// Mitsubishi GX Works2 project: סופי   PLC: FX3G

// global labels: Global1
VAR_GLOBAL
  input_sw AT M0 : BOOL;
  active_day AT M7 : BOOL;
  work_day AT X010 : BOOL;
  flour_stock AT D1100 : REAL;
  flour_input AT D1110 : REAL;
  yeast_stock AT D1120 : REAL;
  oil_stock AT D1160 : REAL;
  spices_stock AT D1180 : REAL;
  yeast_input AT D1130 : REAL;
  water_input AT D1150 : REAL;
  water_stock AT D1140 : REAL;
  oil_input AT D1170 : REAL;
  spices_input AT D1190 : REAL;
  check_flour AT M1 : BOOL;
END_VAR
VAR_GLOBAL CONSTANT
  min_flour_stock : REAL := 100.0;
  yeast_con : REAL := 0.2;
END_VAR
VAR_GLOBAL
  save_mul AT D1200 : REAL;
  check_yeast AT M2 : BOOL;
END_VAR
VAR_GLOBAL CONSTANT
  water_con : REAL := 0.5;
END_VAR
VAR_GLOBAL
  check_water AT M3 : BOOL;
END_VAR
VAR_GLOBAL CONSTANT
  oil_con : REAL := 0.3;
END_VAR
VAR_GLOBAL
  stock_stock AT D1160 : REAL;
  check_oil AT M4 : BOOL;
END_VAR
VAR_GLOBAL CONSTANT
  spices_con : REAL := 0.1;
END_VAR
VAR_GLOBAL
  check_spices AT M5 : BOOL;
  check_stock AT M6 : BOOL;
  emergency_sw AT X007 : BOOL;
END_VAR
VAR_GLOBAL CONSTANT
  flicker_time : INT := 5;
  flicker_con : INT := 6;
  flicker_timer : INT := 30;
  flick_time : INT := 5;
END_VAR
VAR_GLOBAL
  start_dough AT X001 : BOOL;
END_VAR
VAR_GLOBAL CONSTANT
  sec : INT := 30;
END_VAR
VAR_GLOBAL
  end_dough AT TS194 : BOOL;
  dough_light AT Y001 : BOOL;
END_VAR
VAR_GLOBAL CONSTANT
  flour_q : REAL := 100.0;
  yeast_q : REAL := 20.0;
  water_q : REAL := 50.0;
  oil_q : REAL := 30.0;
  spices_q : REAL := 10.0;
END_VAR
VAR_GLOBAL
  active_day_bulb AT Y010 : BOOL;
  start_ingridients_prep AT X002 : BOOL;
  ingridients_light AT Y005 : BOOL;
  start_swell AT X011 : BOOL;
  X11_COUNTER AT CC1 : BOOL;
END_VAR
VAR_GLOBAL CONSTANT
  X11_VAL : INT := 2;
END_VAR
VAR_GLOBAL
  swelling_time AT M8 : BOOL;
  swelling_light_timer AT TC195 : BOOL;
END_VAR
VAR_GLOBAL CONSTANT
  swelling_timer : INT := 30;
END_VAR
VAR_GLOBAL
  blink_light AT M9 : BOOL;
  blink3 AT TC3 : BOOL;
END_VAR
VAR_GLOBAL CONSTANT
  blink_time : INT := 5;
END_VAR
VAR_GLOBAL
  blink_timer3 AT TS3 : BOOL;
  blink_light3 AT Y002 : BOOL;
  blink4 AT TC4 : BOOL;
  blink_timer4 AT TS4 : BOOL;
  blink_light4 AT Y003 : BOOL;
  baking_timer AT TS5 : BOOL;
END_VAR
VAR_GLOBAL CONSTANT
  baking_time : INT := 40;
END_VAR
VAR_GLOBAL
  baking AT TC5 : BOOL;
  baking_light AT Y004 : BOOL;
  sample_quality AT X003 : BOOL;
  analog_input_2 AT D8281 : INT;
  save_analog_input_2 AT D1300 : INT;
END_VAR
VAR_GLOBAL CONSTANT
  lower_analog_bound : INT := K400;
  upper_analog_bound : INT := K2000;
END_VAR
VAR_GLOBAL
  good_quality AT M10 : BOOL;
  move_to_shelves_light AT Y006 : BOOL;
  move_to_shelves AT TC6 : BOOL;
END_VAR
VAR_GLOBAL CONSTANT
  move_to_shelves_time : INT := 50;
END_VAR
VAR_GLOBAL
  move_to_shelves_timer AT TS6 : BOOL;
  failure_counter AT CC2 : BOOL;
END_VAR
VAR_GLOBAL CONSTANT
  failure : INT := 2;
END_VAR
VAR_GLOBAL
  failure_count AT CS2 : BOOL;
  timer_flicker_light AT TC7 : BOOL;
END_VAR
VAR_GLOBAL CONSTANT
  flicker_duration : INT := 30;
END_VAR
VAR_GLOBAL
  timer_flicker1 AT TC8 : BOOL;
END_VAR
VAR_GLOBAL CONSTANT
  flicker_con1 : INT := 5;
END_VAR
VAR_GLOBAL
  timer_flicker2 AT TC9 : BOOL;
  timer_flicker_light_con AT TS7 : BOOL;
  timer_flicker2_con AT TS9 : BOOL;
  timer_flicker1_con AT TS8 : BOOL;
  M_11 AT M11 : BOOL;
  M_12 AT M12 : BOOL;
  flour_container AT D1210 : REAL;
  yeast_container AT D1220 : REAL;
  water_container AT D1230 : REAL;
  oil_container AT D1240 : REAL;
  spices_container AT D1250 : REAL;
  mixer AT D1260 : REAL;
END_VAR
VAR_GLOBAL CONSTANT
  on_sign : REAL := 1.0;
END_VAR
VAR_GLOBAL
  swelling_container AT D1270 : REAL;
  swelling_timer_s AT TS195 : BOOL;
  baking_pan AT D1280 : REAL;
  shelves AT D1290 : REAL;
  is_greater AT M26 : BOOL;
  finish_day AT M30 : BOOL;
  M_31 AT M31 : BOOL;
  M_32 AT M32 : BOOL;
  valid_x11 AT CS1 : BOOL;
  is_lower AT M27 : BOOL;
  finish_iteration AT M40 : BOOL;
  flicker_c AT CC0 : BOOL;
  timer3 AT TC194 : BOOL;
END_VAR

// task Task_01 (event TRUE, interval 0, priority 31): POU_01

PROGRAM POU_01
(* structured ladder/FBD written out as ST: instructions are called as NAME(EN, inputs, outputs); _pN, _eN, _tN stand for wires *)
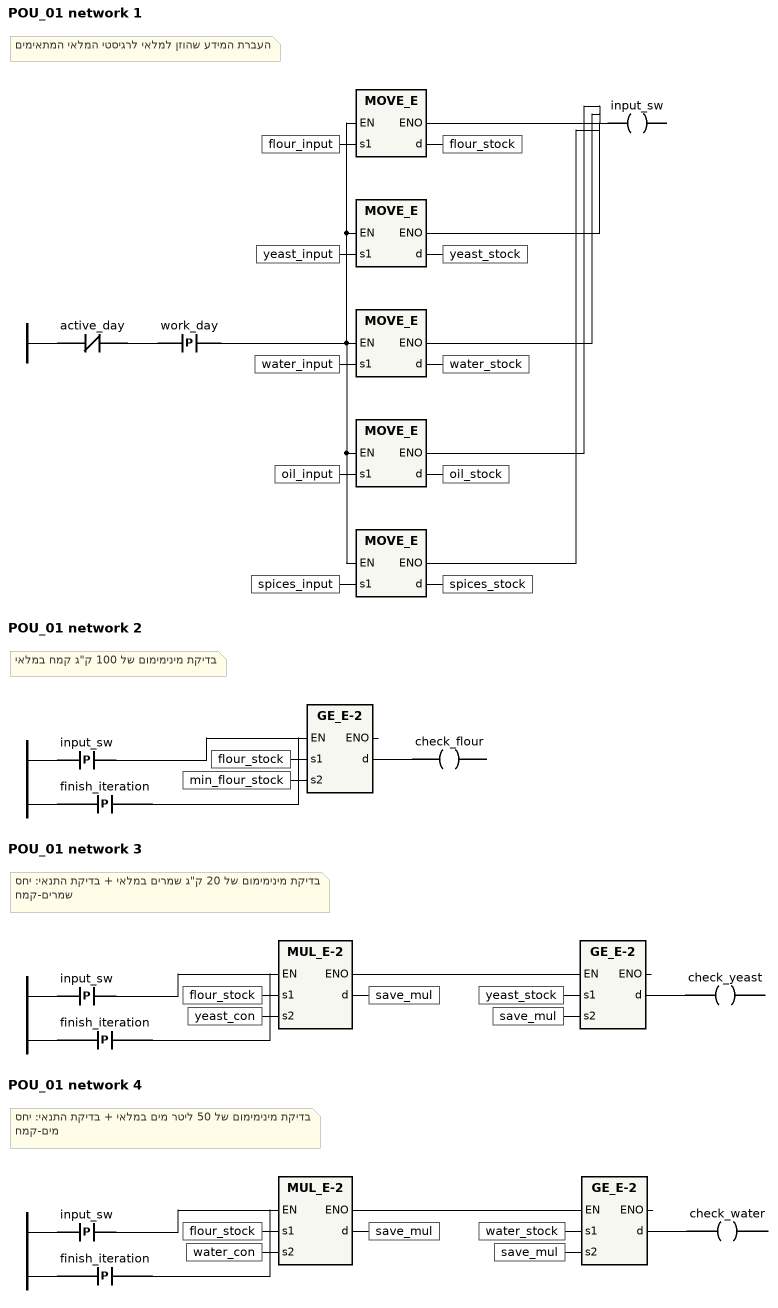
(* network 1 *)
(* העברת המידע שהוזן למלאי לרגיסטי המלאי המתאימים *)
_p1 := NOT active_day AND LDP(TRUE, work_day);
_e2 := MOVE_E(_p1, flour_input, flour_stock);
_e3 := MOVE_E(_p1, yeast_input, yeast_stock);
_e4 := MOVE_E(_p1, water_input, water_stock);
_e5 := MOVE_E(_p1, oil_input, oil_stock);
_e6 := MOVE_E(_p1, spices_input, spices_stock);
input_sw := _e2 OR _e3 OR _e4 OR _e5 OR _e6;
(* network 2 *)
(* בדיקת מינימימום של 100 ק"ג קמח במלאי *)
GE_E(LDP(TRUE, input_sw) OR LDP(TRUE, finish_iteration), flour_stock, min_flour_stock, _t1);
check_flour := _t1;
(* network 3 *)
(* בדיקת מינימימום של 20 ק"ג שמרים במלאי + בדיקת התנאי: יחס שמרים-קמח *)
_e1 := MUL_E(LDP(TRUE, input_sw) OR LDP(TRUE, finish_iteration), flour_stock, yeast_con, save_mul);
GE_E(_e1, yeast_stock, save_mul, _t2);
check_yeast := _t2;
(* network 4 *)
(* בדיקת מינימימום של 50 ליטר מים במלאי + בדיקת התנאי: יחס מים-קמח *)
_e1 := MUL_E(LDP(TRUE, input_sw) OR LDP(TRUE, finish_iteration), flour_stock, water_con, save_mul);
GE_E(_e1, water_stock, save_mul, _t2);
check_water := _t2;
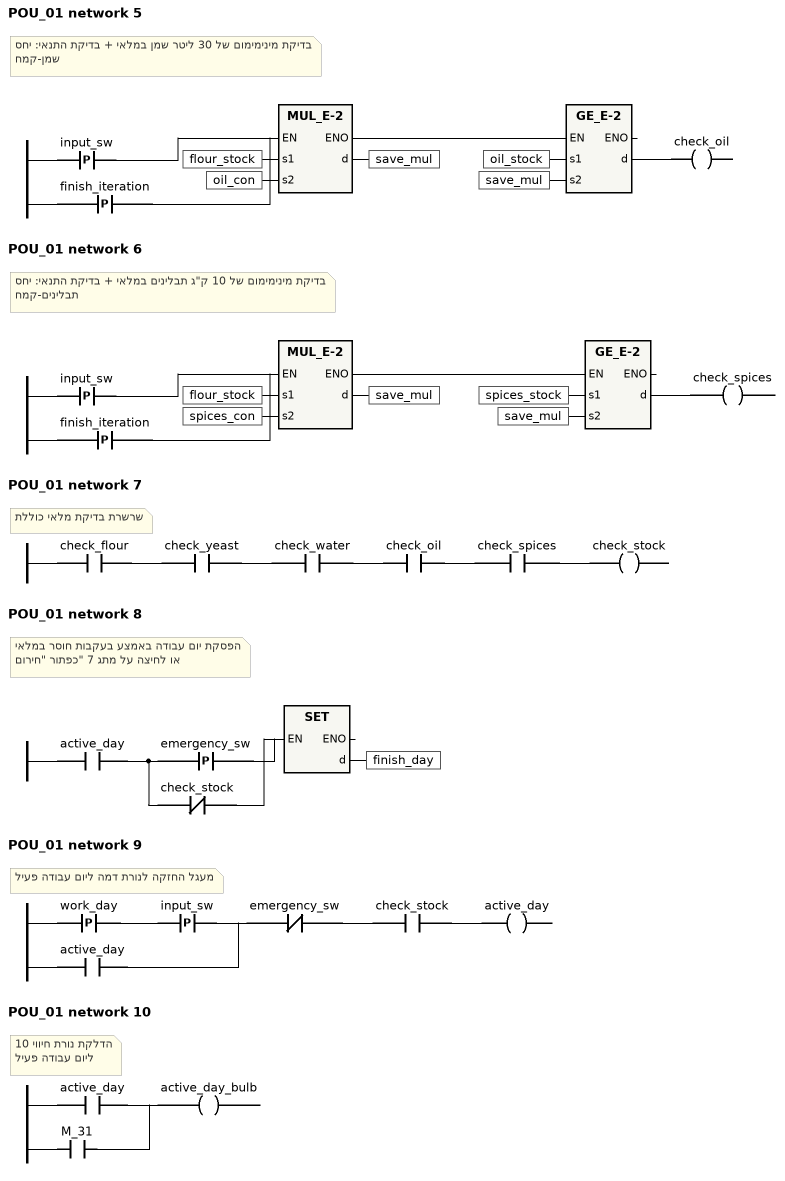
(* network 5 *)
(* בדיקת מינימימום של 30 ליטר שמן במלאי + בדיקת התנאי: יחס שמן-קמח *)
_e1 := MUL_E(LDP(TRUE, input_sw) OR LDP(TRUE, finish_iteration), flour_stock, oil_con, save_mul);
GE_E(_e1, oil_stock, save_mul, _t2);
check_oil := _t2;
(* network 6 *)
(* בדיקת מינימימום של 10 ק"ג תבלינים במלאי + בדיקת התנאי: יחס תבלינים-קמח *)
_e1 := MUL_E(LDP(TRUE, input_sw) OR LDP(TRUE, finish_iteration), flour_stock, spices_con, save_mul);
GE_E(_e1, spices_stock, save_mul, _t2);
check_spices := _t2;
(* network 7 *)
(* שרשרת בדיקת מלאי כוללת *)
check_stock := check_flour AND check_yeast AND check_water AND check_oil AND check_spices;
(* network 8 *)
(* הפסקת יום עבודה באמצע בעקבות חוסר במלאי / או לחיצה על מתג 7 "כפתור "חירום *)
SET((active_day AND LDP(TRUE, emergency_sw)) OR (active_day AND NOT check_stock), finish_day);
(* network 9 *)
(* מעגל החזקה לנורת דמה ליום עבודה פעיל *)
active_day := (((LDP(TRUE, work_day) AND LDP(TRUE, input_sw)) OR active_day) AND NOT emergency_sw) AND check_stock;
(* network 10 *)
(* הדלקת נורת חיווי 10 /  ליום עבודה פעיל *)
active_day_bulb := active_day OR M_31;
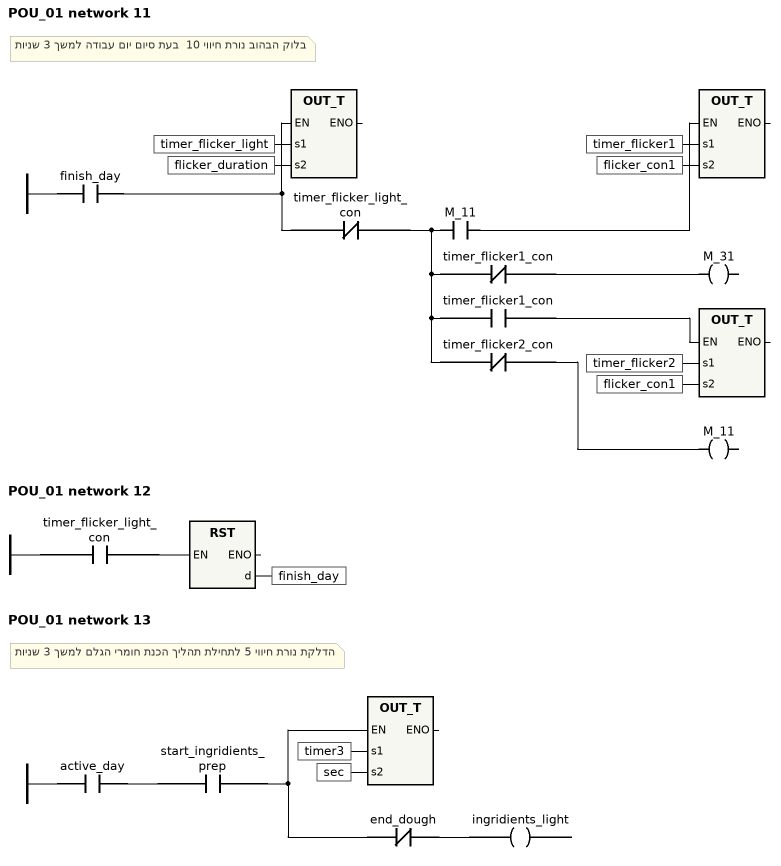
(* network 11 *)
(* בלוק הבהוב נורת חיווי 10  בעת סיום יום עבודה למשך 3 שניות *)
OUT_T(finish_day, timer_flicker_light, flicker_duration);
_p1 := finish_day AND NOT timer_flicker_light_con;
OUT_T(_p1 AND M_11, timer_flicker1, flicker_con1);
M_31 := _p1 AND NOT timer_flicker1_con;
OUT_T(_p1 AND timer_flicker1_con, timer_flicker2, flicker_con1);
M_11 := _p1 AND NOT timer_flicker2_con;
(* network 12 *)
RST(timer_flicker_light_con, finish_day);
(* network 13 *)
(* הדלקת נורת חיווי 5 לתחילת תהליך הכנת חומרי הגלם למשך 3 שניות *)
_p1 := active_day AND start_ingridients_prep;
OUT_T(_p1, timer3, sec);
ingridients_light := _p1 AND NOT end_dough;
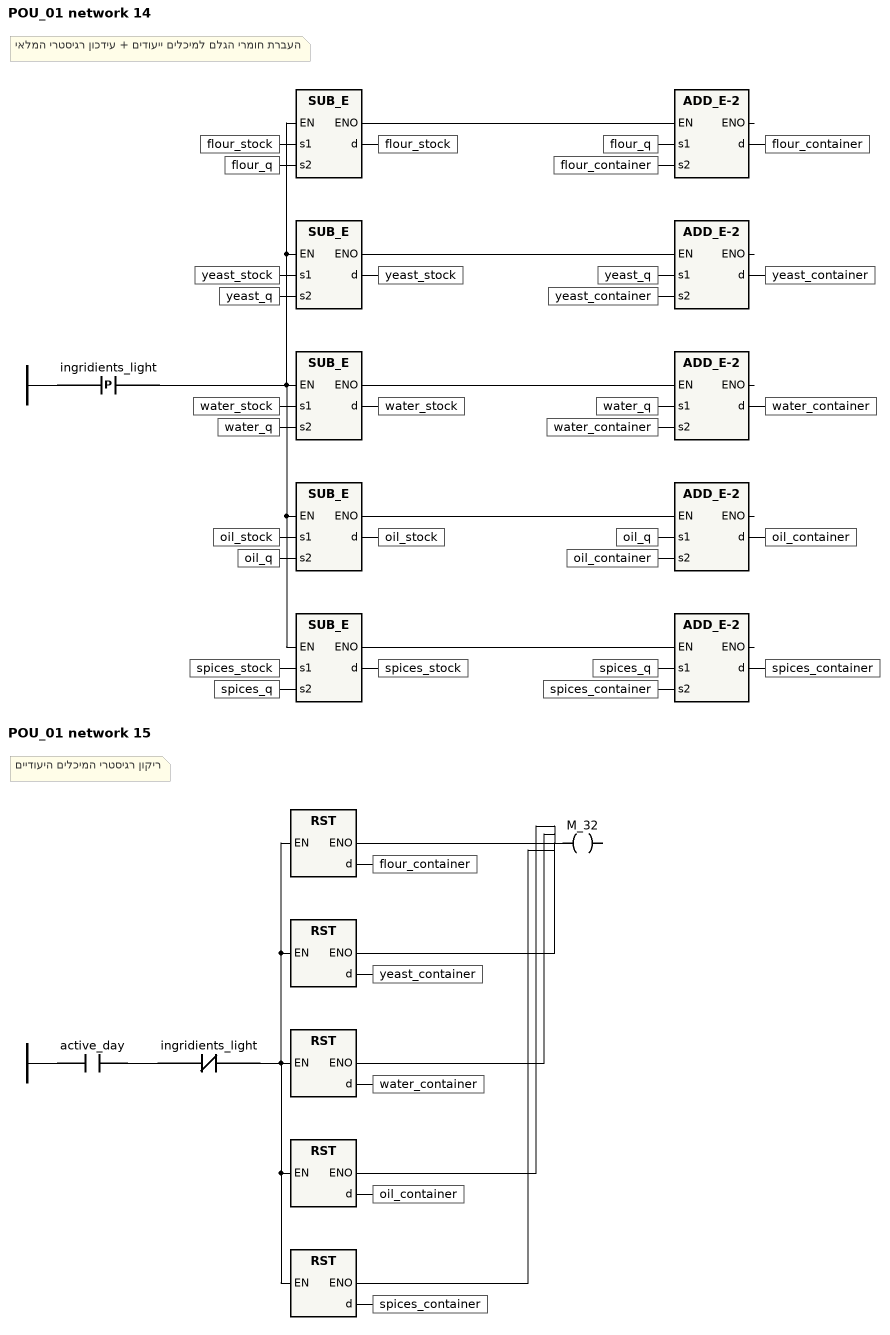
(* network 14 *)
(* העברת חומרי הגלם למיכלים ייעודים + עידכון רגיסטרי המלאי *)
_p1 := LDP(TRUE, ingridients_light);
_e2 := SUB_E(_p1, flour_stock, flour_q, flour_stock);
ADD_E(_e2, flour_q, flour_container, flour_container);
_e3 := SUB_E(_p1, yeast_stock, yeast_q, yeast_stock);
ADD_E(_e3, yeast_q, yeast_container, yeast_container);
_e4 := SUB_E(_p1, water_stock, water_q, water_stock);
ADD_E(_e4, water_q, water_container, water_container);
_e5 := SUB_E(_p1, oil_stock, oil_q, oil_stock);
ADD_E(_e5, oil_q, oil_container, oil_container);
_e6 := SUB_E(_p1, spices_stock, spices_q, spices_stock);
ADD_E(_e6, spices_q, spices_container, spices_container);
(* network 15 *)
(* ריקון רגיסטרי המיכלים היעודיים *)
_p1 := active_day AND NOT ingridients_light;
_e2 := RST(_p1, flour_container);
_e3 := RST(_p1, yeast_container);
_e4 := RST(_p1, water_container);
_e5 := RST(_p1, oil_container);
_e6 := RST(_p1, spices_container);
M_32 := _e2 OR _e3 OR _e4 OR _e5 OR _e6;
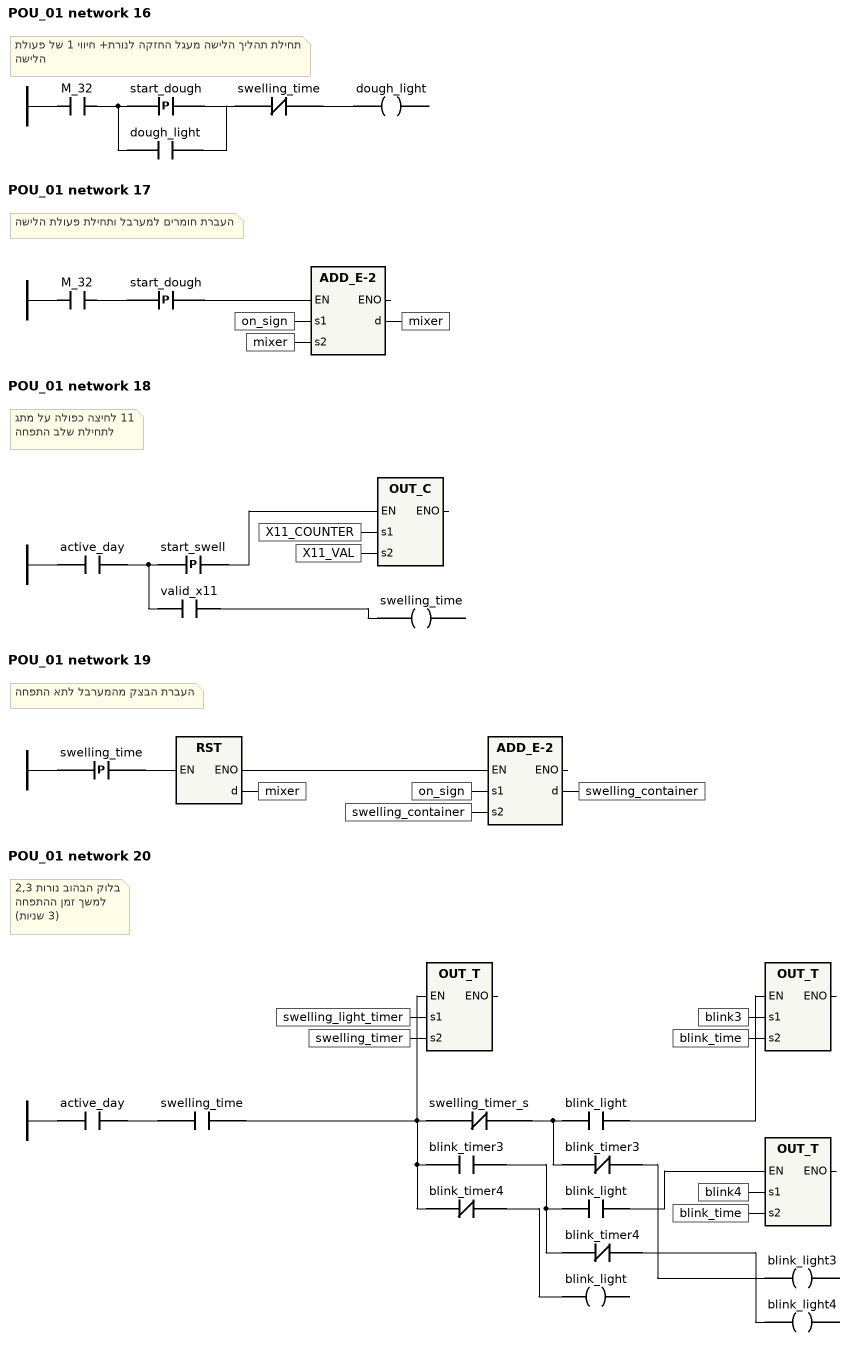
(* network 16 *)
(* תחילת תהליך הלישה מעגל החזקה לנורת+ חיווי 1 של פעולת הלישה *)
dough_light := ((M_32 AND LDP(TRUE, start_dough)) OR (M_32 AND dough_light)) AND NOT swelling_time;
(* network 17 *)
(* העברת חומרים למערבל ותחילת פעולת הלישה *)
ADD_E(M_32 AND LDP(TRUE, start_dough), on_sign, mixer, mixer);
(* network 18 *)
(* 11 לחיצה כפולה על מתג  / לתחילת שלב התפחה *)
OUT_C(active_day AND LDP(TRUE, start_swell), X11_COUNTER, X11_VAL);
swelling_time := active_day AND valid_x11;
(* network 19 *)
(* העברת הבצק מהמערבל לתא התפחה *)
_e1 := RST(LDP(TRUE, swelling_time), mixer);
ADD_E(_e1, on_sign, swelling_container, swelling_container);
(* network 20 *)
(* בלוק הבהוב נורות 2,3 /  למשך זמן ההתפחה /  (3 שניות) *)
_p1 := active_day AND swelling_time;
OUT_T(_p1, swelling_light_timer, swelling_timer);
_p2 := _p1 AND NOT swelling_timer_s;
OUT_T(_p2 AND blink_light, blink3, blink_time);
blink_light3 := _p2 AND NOT blink_timer3;
_p3 := _p1 AND blink_timer3;
OUT_T(_p3 AND blink_light, blink4, blink_time);
blink_light4 := _p3 AND NOT blink_timer4;
blink_light := _p1 AND NOT blink_timer4;
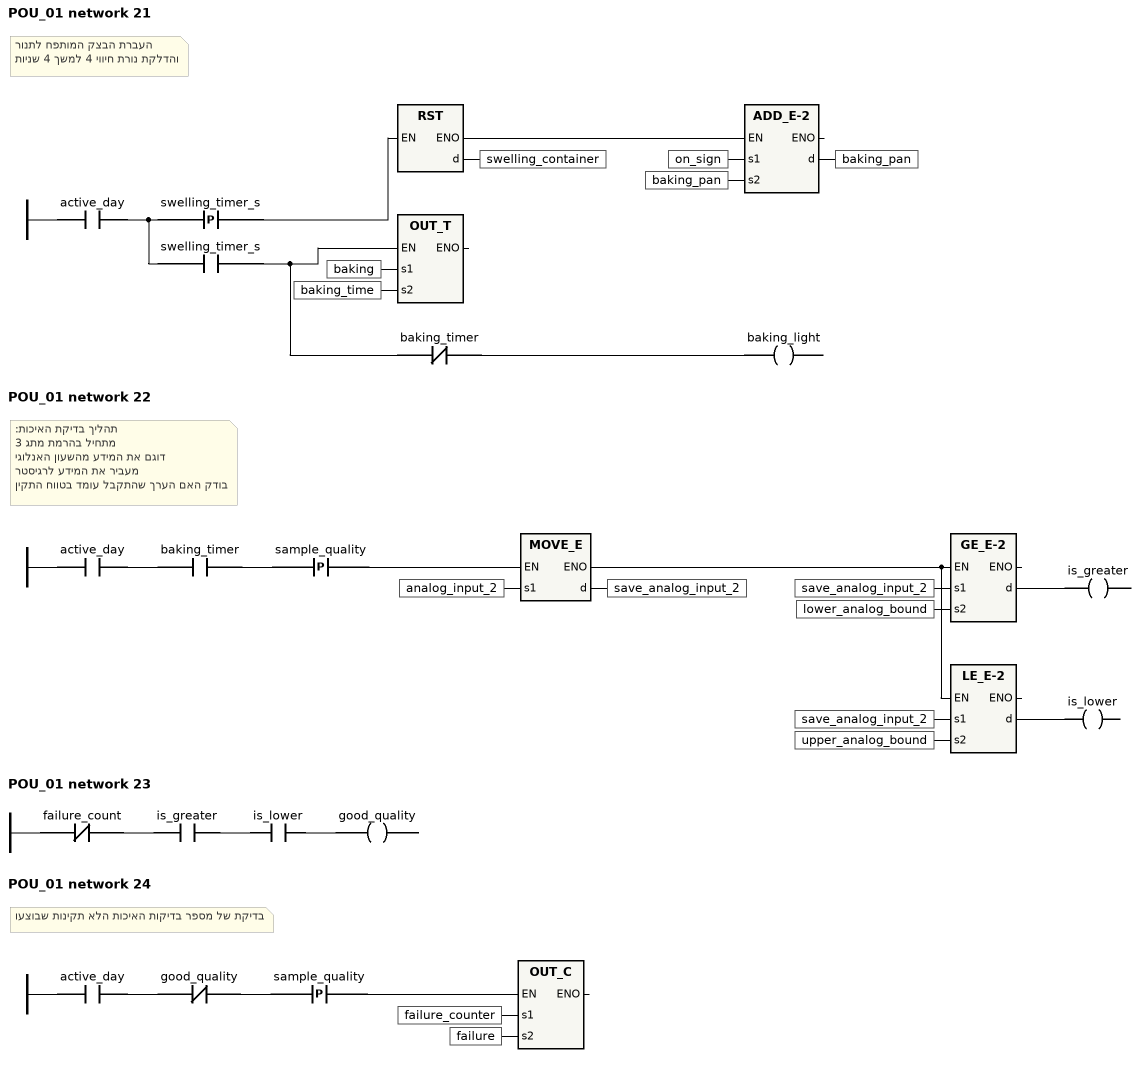
(* network 21 *)
(* העברת הבצק המותפח לתנור   / והדלקת נורת חיווי 4 למשך 4 שניות *)
_e1 := RST(active_day AND LDP(TRUE, swelling_timer_s), swelling_container);
ADD_E(_e1, on_sign, baking_pan, baking_pan);
_p2 := active_day AND swelling_timer_s;
OUT_T(_p2, baking, baking_time);
baking_light := _p2 AND NOT baking_timer;
(* network 22 *)
(* תהליך בדיקת האיכות:  / מתחיל בהרמת מתג 3  / דוגם את המידע מהשעון האנלוגי / מעביר את המידע לרגיסטר / בודק האם הערך שהתקבל עומד בטווח התקין *)
_e1 := MOVE_E(active_day AND baking_timer AND LDP(TRUE, sample_quality), analog_input_2, save_analog_input_2);
GE_E(_e1, save_analog_input_2, lower_analog_bound, _t2);
is_greater := _t2;
LE_E(_e1, save_analog_input_2, upper_analog_bound, _t3);
is_lower := _t3;
(* network 23 *)
good_quality := NOT failure_count AND is_greater AND is_lower;
(* network 24 *)
(* בדיקת של מספר בדיקות האיכות הלא תקינות שבוצעו *)
OUT_C(active_day AND NOT good_quality AND LDP(TRUE, sample_quality), failure_counter, failure);
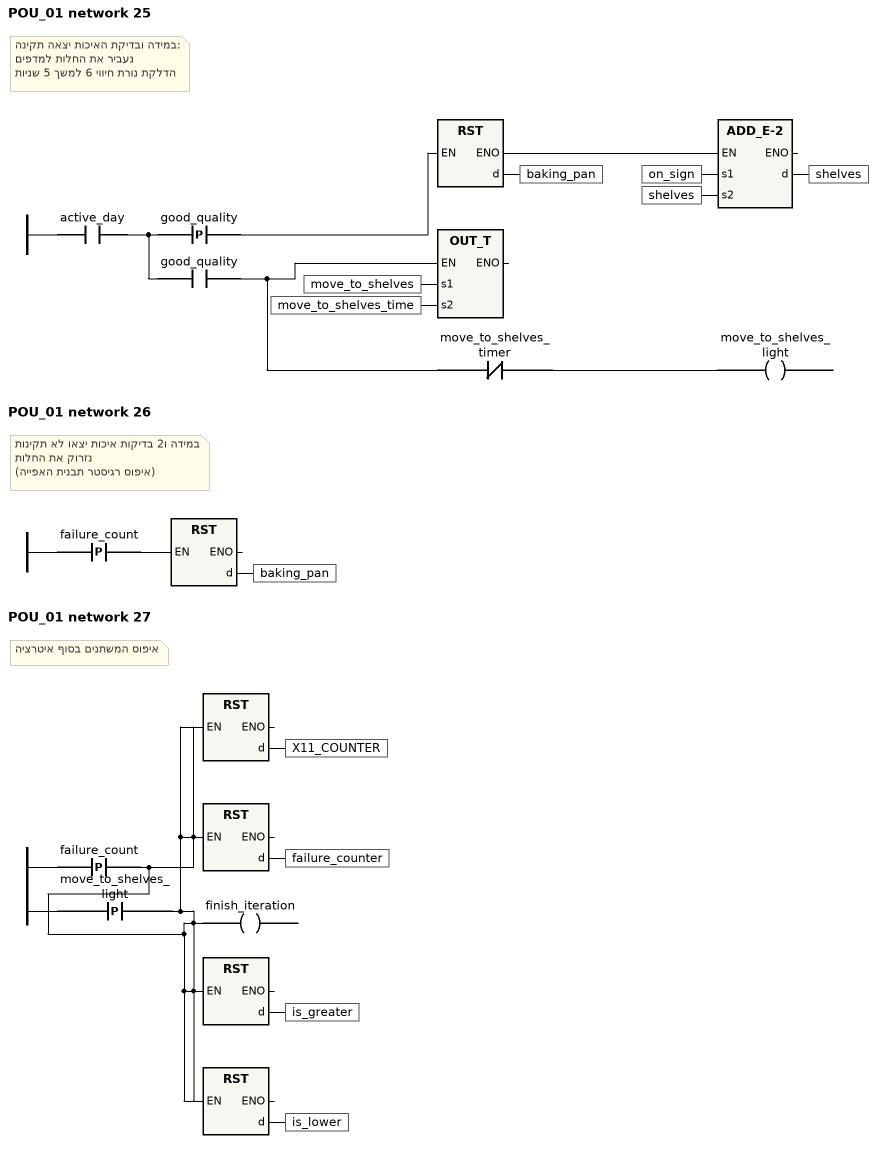
(* network 25 *)
(* :במידה ובדיקת האיכות יצאה תקינה / נעביר את החלות למדפים / הדלקת נורת חיווי 6 למשך 5 שניות *)
_e1 := RST(active_day AND LDP(TRUE, good_quality), baking_pan);
ADD_E(_e1, on_sign, shelves, shelves);
_p2 := active_day AND good_quality;
OUT_T(_p2, move_to_shelves, move_to_shelves_time);
move_to_shelves_light := _p2 AND NOT move_to_shelves_timer;
(* network 26 *)
(* במידה ו2 בדיקות איכות יצאו לא תקינות / נזרוק את החלות  / (איפוס רגיסטר תבנית האפייה) *)
RST(LDP(TRUE, failure_count), baking_pan);
(* network 27 *)
(* איפוס המשתנים בסוף איטרציה *)
_p1 := LDP(TRUE, failure_count) OR LDP(TRUE, move_to_shelves_light);
finish_iteration := _p1;
RST(_p1, X11_COUNTER);
RST(_p1, failure_counter);
RST(_p1, is_greater);
RST(_p1, is_lower);
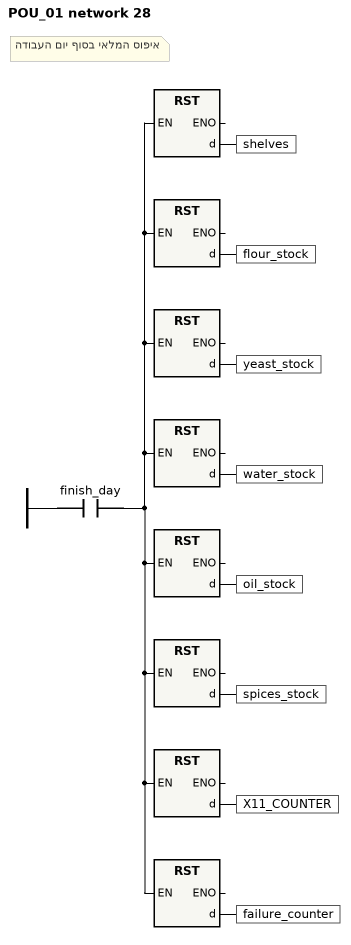
(* network 28 *)
(* איפוס המלאי בסוף יום העבודה *)
RST(finish_day, shelves);
RST(finish_day, flour_stock);
RST(finish_day, yeast_stock);
RST(finish_day, water_stock);
RST(finish_day, oil_stock);
RST(finish_day, spices_stock);
RST(finish_day, X11_COUNTER);
RST(finish_day, failure_counter);
END_PROGRAM
